// TIA Portal V20 export
VAR_GLOBAL   // PLC tag table "LGR_Const_InvalidCode"
END_VAR
VAR_GLOBAL CONSTANT   // user constants
   INVALID_PROTOCOL : UInt := 100;
   INVALID_CMD : UInt := 101;
   INVALID_SRC : UInt := 102;
   INVALID_DST : UInt := 103;
   INVALID_DUPLICATED : UInt := 104;
   INVALID_UNDEFINED : UInt := 900;
   INVALID_TASK_POSX : UInt := 301;
   INVALID_TASK_POSY : UInt := 302;
   INVALID_TASK_POSZ : UInt := 303;
   INVALID_TASK_POSG : UInt := 304;
   INVALID_TASK_TYPE : UInt := 203;
   INVALID_TASK_ITEM_CODE : UInt := 501;
   INVALID_TASK_ITEM_COUNT : UInt := 502;
   INVALID_TASK_BLENDUP : UInt := 310;
   INVALID_TASK_BLENDDOWN : UInt := 311;
   INVALID_TASK_WORKID : UInt := 200;
   INVALID_TASK_TASKID : UInt := 201;
   INVALID_TASK_WORKCELL : UInt := 202;
END_VAR
